{attribute addProperty BoxType "EL3621-0020-0016"}
{attribute addProperty Id "AI_InputsAT %I*AI_Inputs_5C8246304860WcStateAT %I*WcState_F855686C1620InfoDataAT %I*InfoData_BC63D37F80100"}
{attribute addProperty CRC "855316632"}
{attribute addProperty SizeInBites "144"}
{attribute addProperty SizeInBytes "18"}
TYPE EL3621_85E9A035 :
STRUCT
	{attribute addProperty Name "AI_Inputs"}
	AI_Inputs : AI_Inputs_5C824630;
	{attribute addProperty Name "WcState"}
	WcState : WcState_F855686C;
	{attribute addProperty Name "InfoData"}
	InfoData : InfoData_BC63D37F;
END_STRUCT
END_TYPE

(* stored: Version 1.2.0.0, ProductVersion 3.1.4024.9
   DUT EL3621_85E9A035: Id {ff414321-b045-4b76-af8c-07ad069e0246} *)
